{attribute 'GeneratedUsingTerminal: EL3773-0000-0018'}
{attribute addProperty BoxType "EL3773-0000-0018"}
{attribute addProperty Id "I2_StatusAT %I*I2_Status_DC9039207"}
{attribute addProperty CRC "4239878219"}
{attribute addProperty Size "7"}
TYPE L2_Current_Status_FCB7684B :
STRUCT
	{attribute addProperty Name "I2_Status"}
	I2_Status AT %I* : I2_Status_DC903920;
END_STRUCT
END_TYPE

(* stored: Version 1.2.0.0, ProductVersion 3.1.4024.9
   DUT L2_Current_Status_FCB7684B: Id {98e3b35b-9f60-4cc4-8519-c6d641a37bae} *)
